TYPE ST_Batch_HMI :
STRUCT
	bBatchOpen : BOOL;
	bBatchClose : BOOL;
	sBatchName : STRING;
END_STRUCT
END_TYPE

(* stored: Version 1.1.0.1
   DUT ST_Batch_HMI: Id {c5f84415-2fc9-454c-b9bb-788f25e2b126} *)
